Universal Robots PolyScope program: palletsim_to_ur.urp

Program RidzwanPalletSoftware (installation=default directory=/programs/usbdisk/Projects/Palletizing Software Ridzwan createdIn=5.21.2 lastSavedIn=5.21.2 robotSerialNumber=20195500143)
Calibrated DH parameters: a=[0.000205, -0.197852, -0.050148, -0.000026, 0.000123, 0]; d=[0.162569, 168.345858, -323.671776, 155.459333, 0.099845, 0.099705]; alpha=[1.569557, -0.002238, -0.002505, 1.570234, -1.570059, 0]; deltaTheta=[0, -1.087176, 8.812975, -1.442621, 0, 0]
InitVariablesNode
Robot Program (runOnlyOnce=false)
  Script: socket_open("192.168.56.5", 50000,socket_name="socket_0")
  asciiData := socket_read_ascii_float(6,"socket_0",timeout=0)
  MoveJ speed 60 deg/s, acceleration 80 deg/s^2 (useActiveTCP=true optimoveEnabled=false optiMoveSpeed=0.3 optiMoveAcceleration=0.09) feature=Base
    Waypoint Home1: TCP in base x=-138.063 y=-492.113 z=327.658 mm, rx=-0.0047 ry=-3.1382 rz=-0.0078 rad; joints [-90.564, -90.319, -87.209, -92.8, 89.749, -0.222] deg; TCP offset x=0 y=0 z=176.9 mm, rx=0 ry=0 rz=0 rad
    comparisonVar := get_actual_tcp_pose()
  boxCenterX := asciiData[3]
  boxCenterY := asciiData[4]
  CompilePoseRef := p[boxCenterX,boxCenterY,0,0,0,0]
  Mooooove := pose_trans(KhaiRef,CompilePoseRef)
  MoveL speed 250 mm/s, acceleration 1200 mm/s^2 (useActiveTCP=true optimoveEnabled=false optiMoveSpeed=0.3 optiMoveAcceleration=0.09) feature=Base
    Waypoint Variable (Variable): variable=Mooooove
  comparisonVar2 := get_actual_tcp_pose()
  DiffY := comparisonVar[1]-comparisonVar2[1]
  DiffX := comparisonVar2[0]-comparisonVar[0]
  Wait Sleep waitTime=2
  Script: socket_send_string("NEXT", "socket_0")
